PROGRAM JoystickMain
VAR
	
	axDr : AXISdriver;
	btDR : BUTTONdriver;
	ldDr1 : LEDdriver;
	ldDr2 : LEDdriver;
	ldDr3 : LEDdriver;
	calFB : CalibrationFB;
	button : ButtonType := ButtonType.notPressed;
	
	prevStateCal : UINT := 0;
	changeState : BOOL := FALSE;
	
	init : BOOL := TRUE;
	initOp : BOOL := TRUE;
	
	WPDfb : WritePersistentData;
	ShtDNfb : FB_S_UPS_CX51x0;
END_VAR

ShtDNfb(sNetID:='', iPLCPort:=0, iUPSPort:=16#588, tTimeout:=DEFAULT_ADS_TIMEOUT, eUpsMode := eSUPS_ImmediateShutdown);
IF NOT ShtDNfb.bPowerFailDetect THEN


	btDr(buttonChannel := 1);
	btDr.getValue(stateOut => button);
	
	WPDfb();
	
	
	CASE JoystickGVL.state OF
		
		JoystickState.NoCalib:
			IF JoystickGVL.calibration.calibrated = TRUE THEN
				JoystickGVL.state := JoystickState.Operational;
				ldDr1(ledChannel := 1, ledBlink := LEDtype.OFF);//zelena
				//ldDr2(ledChannel := 2, ledBlink := LEDtype.OFF);//rumena
				ldDr3(ledChannel := 3, ledBlink := LEDtype.OFF);//rdeca
			ELSE
				ldDr1(ledChannel := 1, ledBlink := LEDtype.OFF);//zelena
				//ldDr2(ledChannel := 2, ledBlink := LEDtype.OFF);//rumena
				IF init THEN
					ldDr3(ledChannel := 3, ledBlink := LEDtype.OFF);//rdeca
					init := FALSE;
				END_IF
				ldDr3(ledChannel := 3, ledBlink := LEDtype.BlinkContinious, blinkInterval := T#0.2S);//rdeca
				IF button = ButtonType.hold5s THEN
					ldDr1(ledChannel := 1, ledBlink := LEDtype.OFF);//zelena
					ldDr2(ledChannel := 2, ledBlink := LEDtype.OFF);//rumena
					ldDr3(ledChannel := 3, ledBlink := LEDtype.OFF);//rdeca
					JoystickGVL.state := JoystickState.Calib;
				END_IF
			END_IF
				
		JoystickState.Calib:
			
			
			calFB(buttonState := button);
			IF calFB.finished THEN
				JoystickGVL.state := JoystickState.Operational;
				JoystickGVL.calibration := calFB.calibrationParams;
				//save here
				WPDfb(START:=0);
				WPDfb(NETID := '', 	PORT:=801, START:=1, TMOUT := T#1S);
				ldDr1(ledChannel := 1, ledBlink := LEDtype.OFF);//zelena
				//ldDr2(ledChannel := 2, ledBlink := LEDtype.OFF);//rumena
				ldDr3(ledChannel := 3, ledBlink := LEDtype.OFF);//rdeca
			END_IF
			IF calFB.calLight THEN
				ldDR3(ledChannel := 3, ledBLink := LEDtype.OFF);
				ldDR3(ledChannel := 3, ledBLink := LEDtype.BlinkOnce);
			END_IF
			IF calFB.stage1 AND NOT (prevStateCal = 1) THEN
				ldDr1(ledChannel := 1, ledBlink := LEDtype.OFF);//zelena
				//ldDr2(ledChannel := 2, ledBlink := LEDtype.OFF);//rumena
				ldDr3(ledChannel := 3, ledBlink := LEDtype.OFF);//rdeca
				ldDr1(ledChannel := 1, ledBlink := LEDtype.BlinkContinious, blinkInterval := T#1S);//rumena
				prevStateCal := 1;
			ELSIF calFB.stage2 AND NOT (prevStateCal = 2) THEN
				ldDr1(ledChannel := 1, ledBlink := LEDtype.OFF);//zelena
				//ldDr2(ledChannel := 2, ledBlink := LEDtype.OFF);//rumena
				ldDr3(ledChannel := 3, ledBlink := LEDtype.OFF);//rdeca
				//ldDr2(ledChannel := 2, ledBlink := LEDtype.BlinkContinious, blinkInterval := T#0.5S);//rumena
				prevStateCal := 2;
			ELSIF calFB.stage3 AND NOT (prevStateCal = 3) THEN
				ldDr1(ledChannel := 1, ledBlink := LEDtype.OFF);//zelena
				//ldDr2(ledChannel := 2, ledBlink := LEDtype.OFF);//rumena
				ldDr3(ledChannel := 3, ledBlink := LEDtype.OFF);//rdeca
				ldDr1(ledChannel := 1, ledBlink := LEDtype.BlinkContinious, blinkInterval := T#0.2S);//rumena
				prevStateCal := 3;
			ELSE
				ldDr1(ledChannel := 1);//zelena
				//ldDr2(ledChannel := 2);//rumena
				ldDr3(ledChannel := 3);//rdeca
			END_IF
			IF  button = ButtonType.hold5s THEN
				JoystickGVL.state := JoystickState.NoCalib;
				ldDr1(ledChannel := 1, ledBlink := LEDtype.OFF);//zelena
				ldDr2(ledChannel := 2, ledBlink := LEDtype.OFF);//rumena
				ldDr3(ledChannel := 3, ledBlink := LEDtype.OFF);//rdeca
				prevStateCal := 0;
				calFB.reset();
				init := TRUE;
			END_IF
		
		JoystickState.Operational:
			
			IF initOp THEN
				initOp := FALSE;
				JoystickGVL.intState := InternalState.passive;
				ControlGVL.status := ControlGVL.status AND 2#11111111111111111111111111111011;
				ldDr3(ledChannel := 3, ledBlink := LEDtype.OFF);
				//ldDr3(ledChannel := 3, ledBlink := LEDtype.ON);
				ldDr1(ledChannel := 1, ledBlink := LEDtype.OFF);//rumena
				ldDr1(ledChannel := 1, ledBlink := LEDtype.ON);//rumena
				//ldDr2(ledChannel := 2, ledBlink := LEDtype.OFF);//rumena
			END_IF
			ldDr1(ledChannel := 1);
			//ldDr2(ledChannel := 2);
			ldDr3(ledChannel := 3);
			axDR(calibParameters := JoystickGVL.calibration);
			
			JoystickGVL.xSpeed := axDr.xAxis;
			JoystickGVL.ySpeed := axDr.yAxis;
			JoystickGVL.zSpeed := axDr.zAxis;
			
			IF button = ButtonType.pressed AND JoystickGVL.speedScale = 1.0 AND JoystickGVL.intState = InternalState.override THEN
				JoystickGVL.speedScale := 0.5;
				ldDr1(ledChannel := 1, ledBlink := LEDtype.OFF);//rumena
				ldDr1(ledChannel := 1, ledBlink := LEDtype.Pulse, blinkInterval := T#1S);//rumena
			ELSIF button = ButtonType.pressed AND JoystickGVL.speedScale = 0.5 AND JoystickGVL.intState = InternalState.override THEN
				ldDr1(ledChannel := 1, ledBlink := LEDtype.OFF);//rumena
				ldDr1(ledChannel := 1, ledBlink := LEDtype.Pulse, blinkInterval := T#0.5S);//rumena
				JoystickGVL.speedScale := 1.0;
			ELSIF button = ButtonType.hold2s THEN
				//change internal state
				changeState := TRUE;
			ELSIF button = ButtonType.hold5s THEN
				initOp := TRUE;
				JoystickGVL.state := JoystickState.Calib;
				ldDr1(ledChannel := 1, ledBlink := LEDtype.OFF);//zelena
				//ldDr2(ledChannel := 2, ledBlink := LEDtype.OFF);//rumena
				ldDr3(ledChannel := 3, ledBlink := LEDtype.OFF);//rdeca
				prevStateCal := 0;
				calFB.reset();
				init := TRUE;
			END_IF
			
			IF changeState THEN
				changeState := FALSE;
				CASE JoystickGVL.intState OF
					InternalState.override:
						JoystickGVL.intState := InternalState.udpOnly;
						ControlGVL.status := ControlGVL.status AND 2#11111111111111111111111111111101;
						ControlGVL.status := ControlGVL.status OR 2#00000000000000000000000000000100;
						ldDr3(ledChannel := 3, ledBlink := LEDtype.OFF);
						ldDr3(ledChannel := 3, ledBlink := LEDtype.ON);
						ldDr1(ledChannel := 1, ledBlink := LEDtype.OFF);//rumena
						JoystickGVL.speedScale := 0.0;
						JoystickGVL.lastUpdate := TRUE;
					InternalState.passive:
						JoystickGVL.intState := InternalState.override;
						ControlGVL.status := ControlGVL.status OR 2#00000000000000000000000000000010;
						ldDr3(ledChannel := 3, ledBlink := LEDtype.OFF);
						ldDr3(ledChannel := 3, ledBlink := LEDtype.Pulse, blinkInterval := T#0.5S);
						JoystickGVL.speedScale := 0.5;
						ldDr1(ledChannel := 1, ledBlink := LEDtype.OFF);//rumena
						ldDr1(ledChannel := 1, ledBlink := LEDtype.Pulse, blinkInterval := T#1S);//rumena
					InternalState.udpOnly:
						JoystickGVL.intState := InternalState.passive;
						ControlGVL.status := ControlGVL.status AND 2#11111111111111111111111111111011;
						
						ldDr3(ledChannel := 3, ledBlink := LEDtype.OFF);
						//ldDr3(ledChannel := 3, ledBlink := LEDtype.ON);
						ldDr1(ledChannel := 1, ledBlink := LEDtype.OFF);//rumena
						ldDr1(ledChannel := 1, ledBlink := LEDtype.ON);//rumena
						
						JoystickGVL.speedScale := 0.0;
						JoystickGVL.lastUpdate := TRUE;
				END_CASE
			END_IF
			
			IF JoystickGVL.intState = InternalState.udpOnly THEN
				//Udp joystick stuff
				IF JoystickGVL.xSpeed > 0 THEN
					ControlGVL.status := ControlGVL.status OR 2#00000000000000000000000000001000;
				ELSIF JoystickGVL.xSpeed < 0 THEN
					ControlGVL.status := ControlGVL.status OR 2#00000000000000000000000000010000;
				ELSE
					ControlGVL.status := ControlGVL.status AND 2#11111111111111111111111111100111;
				END_IF
				IF JoystickGVL.ySpeed > 0 THEN
					ControlGVL.status := ControlGVL.status OR 2#00000000000000000000000000100000;
				ELSIF JoystickGVL.ySpeed < 0 THEN
					ControlGVL.status := ControlGVL.status OR 2#00000000000000000000000001000000;
				ELSE
					ControlGVL.status := ControlGVL.status AND 2#11111111111111111111111110011111;
				END_IF
				IF JoystickGVL.zSpeed > 0 THEN
					ControlGVL.status := ControlGVL.status OR 2#00000000000000000000000010000000;
				ELSIF JoystickGVL.zSpeed < 0 THEN
					ControlGVL.status := ControlGVL.status OR 2#00000000000000000000000100000000;
				ELSE
					ControlGVL.status := ControlGVL.status AND 2#11111111111111111111111001111111;
				END_IF
				IF button = ButtonType.pressed THEN
					ControlGVL.status := ControlGVL.status OR 2#00000000000000000000001000000000;
				ELSE
					ControlGVL.status := ControlGVL.status AND 2#11111111111111111111110111111111;
				END_IF
			END_IF
			
		
	END_CASE
END_IF

END_PROGRAM

(* stored: Version 1.1.0.1, ProductVersion 3.1.4024.10
   POU JoystickMain: Id {f10c2cc5-948a-4d58-9c5b-d1dfdbbf2cfb}, SpecialFunc None *)
